# EPICS autosave request: support/ebrick/2-2-3/iocBoot/iocebrick/autosave/ebrickQADC.req
$(P)$(R)QADC$(C).SCAN
$(P)$(R)QADC$(C).DESC
$(P)$(R)QADC$(C).PREC
$(P)$(R)QADC$(C).LOPR
$(P)$(R)QADC$(C).HOPR
$(P)$(R)QADC$(C).EGU
